(* PLC project , CODESYS CODESYS V3.5 SP16 Patch 4 *)
(* stored: creationDateTime 2021-04-28T11:44:03.8099099, modificationDateTime 2021-04-28T10:31:29.8104989 *)

FUNCTION_BLOCK ccsSafeCraneNumberSuperv_Test EXTENDS CfUnit.FB_TestSuite
  VAR_INPUT
    in_CraneNoSet1 : WORD;  (* First crane number *)
    in_CraneNoSet2 : WORD;  (* Second crane number *)
  END_VAR
  VAR_OUTPUT
    out_S_CraneNoSupervOk : BOOL;  (* Crane numbers match and are not an empty word *)
    out_S_CraneNo : WORD;  (* A safe crane number. If crane numbers missmatch, this word is set to an empty word *)
  END_VAR
  VAR
    EmptyWord : WORD;
  END_VAR

            FB_CraneNumberSuperv_Test1(); FB_CraneNumberSuperv_Test2(); FB_CraneNumberSuperv_Test3();
          

METHOD FB_CraneNumberSuperv_Test1
  VAR
    Fun : ccsSafeCraneNumberSuperv;
    Result : BOOL;
    ExpectedResult : BOOL := FALSE;
    Condition : BOOL;
  END_VAR
                  TEST('"""+m_name"""');      			      

Fun(in_CraneNoSet1 := """+row[0]+""", in_CraneNoSet2 := """+row[0]+""", out_S_CraneNoSupervOk => Result);    
AssertTrue(Condition := (Result = ExpectedResult),
           Message := 'Result is True');
                                                                                      
TEST_FINISHED();
                
END_METHOD
END_FUNCTION_BLOCK
